{attribute addProperty BoxType "EL2535-0000-0021"}
{attribute addProperty Id "StatusAT %I*Status_F4D34E90162"}
{attribute addProperty CRC "2023135669"}
{attribute addProperty SizeInBites "16"}
{attribute addProperty SizeInBytes "2"}
TYPE PWM_Status_Channel_789699B5 :
STRUCT
	{attribute addProperty Name "Status"}
	Status AT %I* : Status_F4D34E90;
END_STRUCT
END_TYPE

(* stored: Version 1.2.0.0, ProductVersion 3.1.4024.9
   DUT PWM_Status_Channel_789699B5: Id {25fbe357-c63b-4f5e-96ad-de9ca997a4af} *)
